FUNCTION_BLOCK ADD_4 (* Calculate arithmetical sum of magnitude inputs (generic FB) *)
  {SET_ATTRIBUTE(GenericClassName, 'GEN_ADD')}
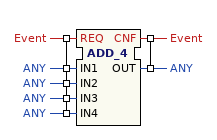
  EVENT_INPUT
    REQ WITH IN1, IN2, IN3, IN4; (* Normal Execution Request *)
  END_EVENT
  EVENT_OUTPUT
    CNF WITH OUT; (* Execution Confirmation *)
  END_EVENT
  VAR_INPUT
    IN1 : ANY; (* ADD input 1 *)
    IN2 : ANY; (* ADD input 2 *)
    IN3 : ANY; (* ADD input 3 *)
    IN4 : ANY; (* ADD input 4 *)
  END_VAR
  VAR_OUTPUT
    OUT : ANY; (* ADD result *)
  END_VAR
END_FUNCTION_BLOCK
